// TIA Portal V17 program export: 0 tag tables, 0 data types, 1 data blocks, 1 code blocks (in call order from the OBs), 0 instance data blocks

DATA_BLOCK "DB_Interface_HMI_Extension"   // DB12
{ S7_Optimized_Access := 'TRUE'; DB_Accessible_From_OPC_UA := 'FALSE' }
AUTHOR : SIEMENS
FAMILY : VW_ADDON
NAME : GENERAL
VERSION : 1.1
// stored: AutoNumber true, DBAccessibleFromOPCUA false, IsOnlyStoredInLoadMemory false, IsRetainMemResEnabled false, IsWriteProtectedInAS false, MemoryReserve 0
   VAR
      BildPanelControl_UhrzeitStellen : Struct   // Screen "Panel Control" Set Date and Time
         EingabeZeit : Date_And_Time := DT#18-5-1-12:0:0.000;   // Eingabe der Uhrzeit und des Datum am Panel im Bild Panel Control / Enter the time and date on the Panel in the Panel Control screen.
         UhrzeitStellen : Bool;   // Übernahme der Uhrzeit und des Datum / Acceptance of time and date
      END_STRUCT;
   END_VAR
BEGIN
END_DATA_BLOCK

ORGANIZATION_BLOCK "OB_Cycle_Extension"   // OB1, LAD, ProgramCycle
TITLE = Cyclic program processing of the VW additional blocks / "Main Program Sweep (Cycle)" / Zyklische Programmbearbeitung der VW Zusatzbausteine
{ S7_Optimized_Access := 'TRUE' }
VERSION : 0.1
// stored: AutoNumber true, IsIECCheckEnabled false, SetENOAutomatically false
   VAR_INPUT
      Initial_Call : Bool;   // Initial call of this OB
      Remanence : Bool;   // =True, if remanent data are available
   END_VAR
   VAR_TEMP
      RET_VAL_WR_LOC_T : Int;
   END_VAR
BEGIN

REGION Network 1: Call FB Machine load and shift model / Aufruf FB Machinenauslastung und Schichtmodell
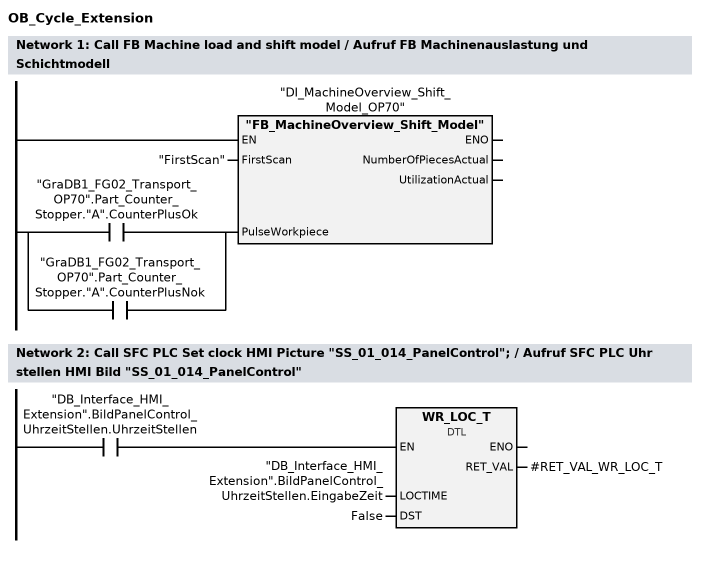
   RUNG wire#powerrail
      "DI_MachineOverview_Shift_Model_OP70"(PulseWorkpiece := wire#w1, FirstScan := "FirstScan", NumberOfPiecesActual =>, UtilizationActual =>)
   END_RUNG
   RUNG wire#powerrail
      Contact( "GraDB1_FG02_Transport_OP70".Part_Counter_Stopper."A".CounterPlusOk )
   END_RUNG wire#w1
   RUNG wire#powerrail
      Contact( "GraDB1_FG02_Transport_OP70".Part_Counter_Stopper."A".CounterPlusNok )
   END_RUNG wire#w1
   // the same network as SCL:
   "DI_MachineOverview_Shift_Model_OP70"(FirstScan := "FirstScan",   // "FB_MachineOverview_Shift_Model"
                           PulseWorkpiece := "GraDB1_FG02_Transport_OP70".Part_Counter_Stopper."A".CounterPlusOk OR "GraDB1_FG02_Transport_OP70".Part_Counter_Stopper."A".CounterPlusNok);
END_REGION

REGION Network 2: Call SFC PLC Set clock HMI Picture "SS_01_014_PanelControl"; / Aufruf SFC PLC Uhr stellen HMI Bild "SS_01_014_PanelControl"
   RUNG wire#powerrail
      Contact( "DB_Interface_HMI_Extension".BildPanelControl_UhrzeitStellen.UhrzeitStellen )
      { S7_Templates := "loctime_type := DTL" } WR_LOC_T(LOCTIME := "DB_Interface_HMI_Extension".BildPanelControl_UhrzeitStellen.EingabeZeit, DST := False, Ret_Val => #RET_VAL_WR_LOC_T)
   END_RUNG
   // the same network as SCL:
   IF "DB_Interface_HMI_Extension".BildPanelControl_UhrzeitStellen.UhrzeitStellen THEN
       #RET_VAL_WR_LOC_T := WR_LOC_T(LOCTIME := "DB_Interface_HMI_Extension".BildPanelControl_UhrzeitStellen.EingabeZeit,
                               DST := False);
   END_IF;
END_REGION
END_ORGANIZATION_BLOCK
